// TIA Portal project "SDRIVELEARN" (V17)

(* hardware
DEVICE "SINAMICS G_1"  Sinamics.Device
   slot 0: "Drive_1"  G120 CU250S-2 PN Vector  6SL3246-0BA22-1FA0  4.7.13
      slot 1: "PROFINET interface"  MDD-SinamicsG120-P
   slot 0: "	_0"  Rail  SinamicsG120SVecto
   slot 3: "PM240 IP20"  PM240 IP20  6SL3224-0BE17-5UA0  -
DEVICE "S7-1200 station_1"  S7-1200 Station
   slot 0: "Rack_0"  S7-1200 Rack  Rack  V1.0
   slot 1: "PLC_1"  CPU 1214C DC/DC/DC  6ES7 214-1AG40-0XB0  V4.2
*)

// ===== PLC "PLC_1"  CPU 1214C DC/DC/DC =====

ORGANIZATION_BLOCK "Main"   // OB1, LAD, ProgramCycle
TITLE = "Main Program Sweep (Cycle)"
{ S7_Optimized_Access := 'TRUE' }
VERSION : 0.1
   VAR_INPUT
      Initial_Call : Bool;   // Initial call of this OB
      Remanence : Bool;   // =True, if remanent data are available
   END_VAR
BEGIN
END_ORGANIZATION_BLOCK